// Mitsubishi GX Works2 project: 실린더 제어하기2-2 0920   PLC: Q03UDV

PROGRAM MAIN
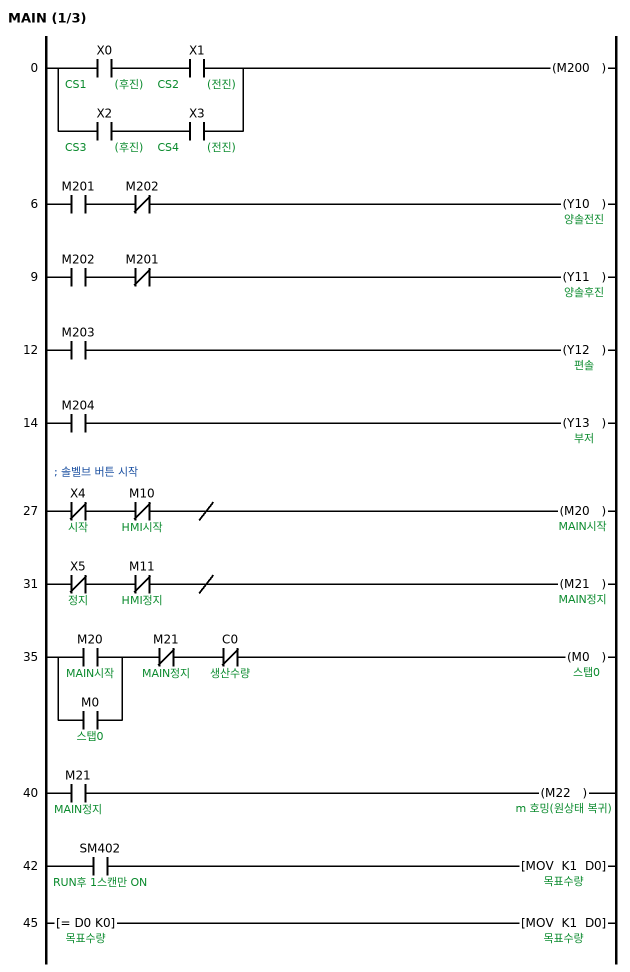
0     LD      X0  ; CS1        (후진)
      AND     X1  ; CS2        (전진)
      LD      X2  ; CS3        (후진)
      AND     X3  ; CS4        (전진)
      ORB
      OUT     M200
6     LD      M201
      ANI     M202
      OUT     Y10  ; 양솔전진
9     LD      M202
      ANI     M201
      OUT     Y11  ; 양솔후진
12    LD      M203
      OUT     Y12  ; 편솔
14    LD      M204
      OUT     Y13  ; 부저
; 솔벨브 버튼 시작
27    LDI     X4  ; 시작
      ANI     M10  ; HMI시작
      INV
      OUT     M20  ; MAIN시작
31    LDI     X5  ; 정지
      ANI     M11  ; HMI정지
      INV
      OUT     M21  ; MAIN정지
35    LD      M20  ; MAIN시작
      OR      M0  ; 스탭0
      ANI     M21  ; MAIN정지
      ANI     C0  ; 생산수량
      OUT     M0  ; 스탭0
40    LD      M21  ; MAIN정지
      OUT     M22  ; m 호밍(원상태 복귀)
42    LD      SM402  ; RUN후 1스캔만 ON
      MOV     K1 D0  ; 목표수량
45    LD=     D0 K0  ; 목표수량
      MOV     K1 D0
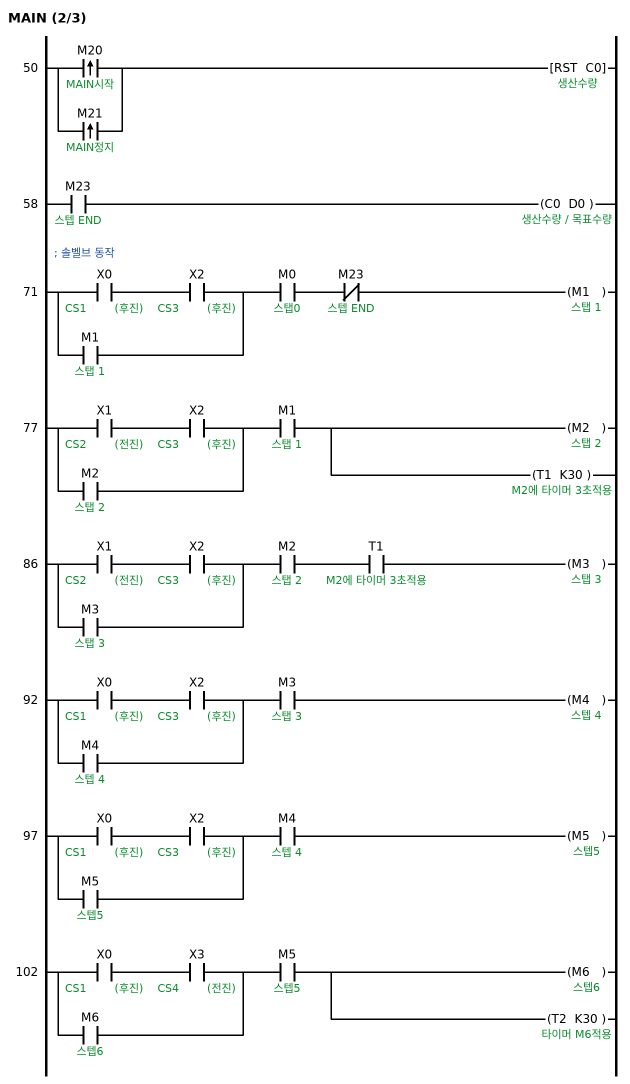
50    LDP     M20  ; MAIN시작
      ORP     M21  ; MAIN정지
      RST     C0  ; 생산수량
58    LD      M23  ; 스텝 END
      OUT     C0 D0  ; 생산수량 / 목표수량
; 솔벨브 동작
71    LD      X0  ; CS1        (후진)
      AND     X2  ; CS3        (후진)
      OR      M1  ; 스탭 1
      AND     M0  ; 스탭0
      ANI     M23  ; 스텝 END
      OUT     M1  ; 스탭 1
77    LD      X1  ; CS2        (전진)
      AND     X2  ; CS3        (후진)
      OR      M2  ; 스탭 2
      AND     M1  ; 스탭 1
      OUT     M2  ; 스탭 2
      OUT     T1 K30  ; M2에 타이머 3초적용
86    LD      X1  ; CS2        (전진)
      AND     X2  ; CS3        (후진)
      OR      M3  ; 스탭 3
      AND     M2  ; 스탭 2
      AND     T1  ; M2에 타이머 3초적용
      OUT     M3  ; 스탭 3
92    LD      X0  ; CS1        (후진)
      AND     X2  ; CS3        (후진)
      OR      M4  ; 스텝 4
      AND     M3  ; 스탭 3
      OUT     M4  ; 스텝 4
97    LD      X0  ; CS1        (후진)
      AND     X2  ; CS3        (후진)
      OR      M5  ; 스텝5
      AND     M4  ; 스텝 4
      OUT     M5  ; 스텝5
102   LD      X0  ; CS1        (후진)
      AND     X3  ; CS4        (전진)
      OR      M6  ; 스텝6
      AND     M5  ; 스텝5
      OUT     M6  ; 스텝6
      OUT     T2 K30  ; 타이머 M6적용
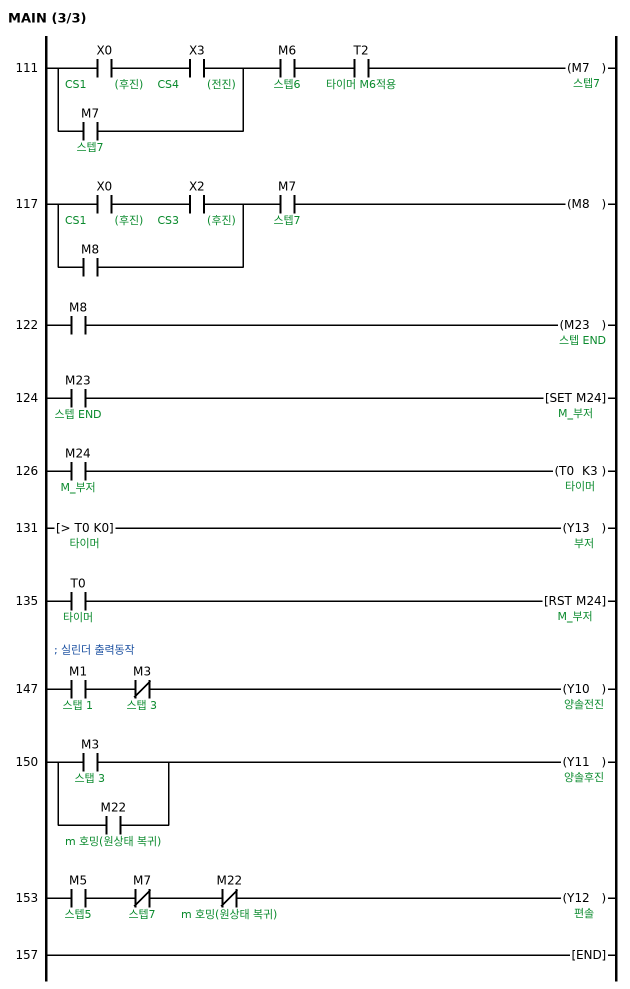
111   LD      X0  ; CS1        (후진)
      AND     X3  ; CS4        (전진)
      OR      M7  ; 스텝7
      AND     M6  ; 스텝6
      AND     T2  ; 타이머 M6적용
      OUT     M7  ; 스텝7
117   LD      X0  ; CS1        (후진)
      AND     X2  ; CS3        (후진)
      OR      M8
      AND     M7  ; 스텝7
      OUT     M8
122   LD      M8
      OUT     M23  ; 스텝 END
124   LD      M23  ; 스텝 END
      SET     M24  ; M_부저
126   LD      M24  ; M_부저
      OUT     T0 K3  ; 타이머
131   LD>     T0 K0  ; 타이머
      OUT     Y13  ; 부저
135   LD      T0  ; 타이머
      RST     M24  ; M_부저
; 실린더 출력동작
147   LD      M1  ; 스탭 1
      ANI     M3  ; 스탭 3
      OUT     Y10  ; 양솔전진
150   LD      M3  ; 스탭 3
      OR      M22  ; m 호밍(원상태 복귀)
      OUT     Y11  ; 양솔후진
153   LD      M5  ; 스텝5
      ANI     M7  ; 스텝7
      ANI     M22  ; m 호밍(원상태 복귀)
      OUT     Y12  ; 편솔
157   END
END_PROGRAM

// device comments not shown above
M25  ; 부저
